FUNCTION_BLOCK FB_System_RND_HVAC
VAR_IN_OUT
	// Hold a reference to MBMaster - may need to share this with other dosing machines if only 1 x RS485 card is used for both
	{attribute 'OPC.UA.DA' := '0'}
  	{attribute 'OPC.UA.DA.StructuredType' := '0'}
	fbModbusManager: 	FB_ModbusManager;    // We can read 32 registers using one query
END_VAR

VAR
	bFirstRun: BOOL := TRUE;
	bResetTimer: BOOL := TRUE;
	tgModReadAdaptorStatus: R_TRIG;
	
	
	nModbusID: INT := 1;
	nNumberHVACUnits: INT := 13;
	
	stModReadAdaptorStatus: 				ST_Modbus_ReadRequest;
	
	stModReadIndoorUnitConnStatus: 			ST_Modbus_ReadRequest;
	stModReadIndoorUnitCommsStatus: 		ST_Modbus_ReadRequest;
	stModReadIndoorUnitSetpoits: 			ARRAY[1..13] OF ST_Modbus_ReadRequest;
	stModReadIndoorUnitPower: 				ARRAY[1..13] OF ST_Modbus_ReadRequest;
	
	stModWriteaAdaptorStatus:				ST_Modbus_WriteRequest;
	stModWriteIndoorRoom:					ST_Modbus_WriteRequest;
	stModWriteIndoorSetpoint_R6:			ST_Modbus_WriteRequest;
	stModWriteIndoorSetpoint_R7:			ST_Modbus_WriteRequest;
	stModWriteIndoorSetpoint_R8:			ST_Modbus_WriteRequest;
	stModWriteIndoorSetpoint_R9:			ST_Modbus_WriteRequest;
	stModWriteIndoorControlPower:			ARRAY[1..13] OF ST_Modbus_WriteRequest;
	stModWriteIndoorControlSetpoint:		ARRAY[1..13] OF ST_Modbus_WriteRequest;
	
	bRoom7or9: BOOL := FALSE;
	nRoomNumber: UINT := 6;
	
	fbTON_DataRefresh: TON := (PT := T#1m, IN := FALSE);
	
	// delete this after commissioning (used for testing)
	modWrite: R_TRIG;
	stModWrite: ST_Modbus_WriteRequest;
	
		// delete this after commissioning (used for testing)
	modRead: 	R_TRIG;
	stModRead: 	ST_Modbus_ReadRequest;
END_VAR

VAR_OUTPUT
	{attribute 'OPC.UA.DA' := '1'}
  	{attribute 'OPC.UA.DA.StructuredType' := '1'}
	fbRND_HVAC: ARRAY[1..13] OF FB_HVAC_RND_Indoor_Unit;
	
	
	i: INT := 0;
	
END_VAR

IF bFirstRun THEN
	devices_init();
	bFirstRun := FALSE;
	initModRequests();
	
	fbModbusManager.addRequest_Write(WriteRequest := ADR(stModWriteaAdaptorStatus));
	fbModbusManager.addRequest_Write(WriteRequest := ADR(stModWriteIndoorRoom));
END_IF

IF bResetTimer THEN
	fbTON_DataRefresh(IN := TRUE);
	bResetTimer := FALSE;
END_IF

fbTON_DataRefresh();
scanInputs();

IF fbTON_DataRefresh.Q THEN
	//fbModbusManager.addRequest_Read(ReadRequest := ADR(stModReadAdaptorStatus));
	//fbModbusManager.addRequest_Read(ReadRequest := ADR(stModReadIndoorUnitConnStatus));
	//fbModbusManager.addRequest_Read(ReadRequest := ADR(stModReadIndoorUnitCommsStatus));
	CASE nRoomNumber OF
		6:
			stModWriteIndoorSetpoint_R6.WriteRegVals[1] := INT_TO_WORD(REAL_TO_INT(Inputs.HVAC_RND[6].Setpoint * 10));
			fbModbusManager.addRequest_Write(WriteRequest := ADR(stModWriteIndoorSetpoint_R6));		
			nRoomNumber := 7;
	
		7:
			stModWriteIndoorSetpoint_R7.WriteRegVals[1] := INT_TO_WORD(REAL_TO_INT(Inputs.HVAC_RND[7].Setpoint * 10));
			fbModbusManager.addRequest_Write(WriteRequest := ADR(stModWriteIndoorSetpoint_R7));
			nRoomNumber := 8;
			
		8:
			stModWriteIndoorSetpoint_R8.WriteRegVals[1] := INT_TO_WORD(REAL_TO_INT(Inputs.HVAC_RND[8].Setpoint * 10));
			fbModbusManager.addRequest_Write(WriteRequest := ADR(stModWriteIndoorSetpoint_R8));
			nRoomNumber := 9;	
		
		9:
			stModWriteIndoorSetpoint_R9.WriteRegVals[1] := INT_TO_WORD(REAL_TO_INT(Inputs.HVAC_RND[9].Setpoint * 10));
			fbModbusManager.addRequest_Write(WriteRequest := ADR(stModWriteIndoorSetpoint_R9));
			nRoomNumber := 6;		
			
	END_CASE
	
	(*
	IF bRoom7or9 THEN
			stModWriteIndoorSetpoint_R7.WriteRegVals[1] := INT_TO_WORD(REAL_TO_INT(Inputs.HVAC_RND[7].Setpoint * 10));
			fbModbusManager.addRequest_Write(WriteRequest := ADR(stModWriteIndoorSetpoint_R7));
			bRoom7or9 := FALSE;
	ELSE
			stModWriteIndoorSetpoint_R9.WriteRegVals[1] := INT_TO_WORD(REAL_TO_INT(Inputs.HVAC_RND[9].Setpoint * 10));
			fbModbusManager.addRequest_Write(WriteRequest := ADR(stModWriteIndoorSetpoint_R9));
			bRoom7or9 := TRUE;
	END_IF
	*)

	

	
	//FOR i := 1 TO 13 DO
		//fbModbusManager.addRequest_Read(ReadRequest := ADR(stModReadIndoorUnitSetpoits[i]));
		//fbModbusManager.addRequest_Read(ReadRequest := ADR(stModReadIndoorUnitPower[i]));
		//fbModbusManager.addRequest_Write(WriteRequest := ADR(stModWriteIndoorControlPower));
		//fbModbusManager.addRequest_Write(WriteRequest := ADR(stModWriteIndoorControlSetpoint));
	//END_FOR
	
	fbTON_DataRefresh(IN := FALSE);
	bResetTimer := TRUE;
END_IF


modRead();
IF modRead.Q THEN
	fbModbusManager.addRequest_Read_Priority(ReadRequest := ADR(stModRead));
END_IF


modWrite();
IF modWrite.Q THEN
	fbModbusManager.addRequest_Write(WriteRequest := ADR(stModWrite));
END_IF

devices_update();

METHOD devices_init : BOOL
VAR_INPUT
END_VAR
(*
aHVAC_IndoorUnits[1] := ADR(fbRND1_HVAC);
aHVAC_IndoorUnits[2] := ADR(fbRND2_HVAC);
aHVAC_IndoorUnits[3] := ADR(fbRND3_HVAC);
aHVAC_IndoorUnits[4] := ADR(fbRND4_HVAC);
aHVAC_IndoorUnits[5] := ADR(fbRND5_HVAC);
aHVAC_IndoorUnits[6] := ADR(fbRND6_HVAC);
aHVAC_IndoorUnits[7] := ADR(fbRND7_HVAC);
aHVAC_IndoorUnits[8] := ADR(fbRND8_HVAC);
aHVAC_IndoorUnits[9] := ADR(fbRND9_HVAC);
aHVAC_IndoorUnits[10] := ADR(fbRND10_HVAC);
aHVAC_IndoorUnits[11] := ADR(fbRND11_HVAC);
aHVAC_IndoorUnits[12] := ADR(fbRND12_HVAC);

*)
END_METHOD

METHOD devices_update : BOOL
VAR_INPUT
END_VAR
(*
FOR i := 1 TO 13 DO
	fbRND_HVAC[i].bOnOff_1_0 := 	stModReadIndoorUnitPower[i].ReadRegsVals[1].0;
	fbRND_HVAC[1].nSetpoint_RO := 	WORD_TO_REAL(stModReadIndoorUnitSetpoits[i].ReadRegsVals[1])/10;
	
END_FOR

fbRND_HVAC[1].bConnectionStatus := stModReadIndoorUnitConnStatus.ReadRegsVals[1].0;
fbRND_HVAC[2].bConnectionStatus := stModReadIndoorUnitConnStatus.ReadRegsVals[1].1;
fbRND_HVAC[3].bConnectionStatus := stModReadIndoorUnitConnStatus.ReadRegsVals[1].2;
fbRND_HVAC[4].bConnectionStatus := stModReadIndoorUnitConnStatus.ReadRegsVals[1].3;
fbRND_HVAC[5].bConnectionStatus := stModReadIndoorUnitConnStatus.ReadRegsVals[1].4;
fbRND_HVAC[6].bConnectionStatus := stModReadIndoorUnitConnStatus.ReadRegsVals[1].5;
fbRND_HVAC[7].bConnectionStatus := stModReadIndoorUnitConnStatus.ReadRegsVals[1].6;
fbRND_HVAC[8].bConnectionStatus := stModReadIndoorUnitConnStatus.ReadRegsVals[1].7;
fbRND_HVAC[9].bConnectionStatus := stModReadIndoorUnitConnStatus.ReadRegsVals[1].8;
fbRND_HVAC[10].bConnectionStatus := stModReadIndoorUnitConnStatus.ReadRegsVals[1].9;
fbRND_HVAC[11].bConnectionStatus := stModReadIndoorUnitConnStatus.ReadRegsVals[1].10;
fbRND_HVAC[12].bConnectionStatus := stModReadIndoorUnitConnStatus.ReadRegsVals[1].11;
fbRND_HVAC[13].bConnectionStatus := stModReadIndoorUnitConnStatus.ReadRegsVals[1].12;

fbRND_HVAC[1].bCommsStatus := stModReadIndoorUnitCommsStatus.ReadRegsVals[1].0;
fbRND_HVAC[2].bCommsStatus := stModReadIndoorUnitCommsStatus.ReadRegsVals[1].1;
fbRND_HVAC[3].bCommsStatus := stModReadIndoorUnitCommsStatus.ReadRegsVals[1].2;
fbRND_HVAC[4].bCommsStatus := stModReadIndoorUnitCommsStatus.ReadRegsVals[1].3;
fbRND_HVAC[5].bCommsStatus := stModReadIndoorUnitCommsStatus.ReadRegsVals[1].4;
fbRND_HVAC[6].bCommsStatus := stModReadIndoorUnitCommsStatus.ReadRegsVals[1].5;
fbRND_HVAC[7].bCommsStatus := stModReadIndoorUnitCommsStatus.ReadRegsVals[1].6;
fbRND_HVAC[8].bCommsStatus := stModReadIndoorUnitCommsStatus.ReadRegsVals[1].7;
fbRND_HVAC[9].bCommsStatus := stModReadIndoorUnitCommsStatus.ReadRegsVals[1].8;
fbRND_HVAC[10].bCommsStatus := stModReadIndoorUnitCommsStatus.ReadRegsVals[1].9;
fbRND_HVAC[11].bCommsStatus := stModReadIndoorUnitCommsStatus.ReadRegsVals[1].10;
fbRND_HVAC[12].bCommsStatus := stModReadIndoorUnitCommsStatus.ReadRegsVals[1].11;
fbRND_HVAC[13].bCommsStatus := stModReadIndoorUnitCommsStatus.ReadRegsVals[1].12;
*)
END_METHOD

METHOD FB_init : BOOL
VAR_INPUT
	bInitRetains : BOOL; // if TRUE, the retain variables are initialized (warm start / cold start)
	bInCopyCode : BOOL;  // if TRUE, the instance afterwards gets moved into the copy code (online change)
	
	ModbusID: UINT;
END_VAR
nModbusID := ModbusID;
END_METHOD

METHOD initModRequests : BOOL
VAR_INPUT
END_VAR

stModReadAdaptorStatus.SlaveAddress := 1;
stModReadAdaptorStatus.AdrFirstSlaveRegisterRead := 0;
stModReadAdaptorStatus.QtyWordsToRead := 1;

stModReadIndoorUnitConnStatus.SlaveAddress := 1;
stModReadIndoorUnitConnStatus.AdrFirstSlaveRegisterRead := 1;
stModReadIndoorUnitConnStatus.QtyWordsToRead := 1;

stModReadIndoorUnitCommsStatus.SlaveAddress := 1;
stModReadIndoorUnitCommsStatus.AdrFirstSlaveRegisterRead := 5;
stModReadIndoorUnitCommsStatus.QtyWordsToRead := 1;

stModWriteaAdaptorStatus.SlaveAddress := 1;
stModWriteaAdaptorStatus.AdrFirstSlaveRegisterWrite := 1;
stModWriteaAdaptorStatus.QtyWordsToWrite := 1;
stModWriteaAdaptorStatus.WriteRegVals[1] := 32768; // turn modbus comms on

stModWriteIndoorRoom.SlaveAddress := 1;
stModWriteIndoorRoom.AdrFirstSlaveRegisterWrite := 2018;
stModWriteIndoorRoom.QtyWordsToWrite := 1;
stModWriteIndoorRoom.WriteRegVals[1] := 1889;

stModWriteIndoorSetpoint_R6.SlaveAddress := 1;
stModWriteIndoorSetpoint_R6.AdrFirstSlaveRegisterWrite := 2017;
stModWriteIndoorSetpoint_R6.QtyWordsToWrite := 1;

stModWriteIndoorSetpoint_R7.SlaveAddress := 1;
stModWriteIndoorSetpoint_R7.AdrFirstSlaveRegisterWrite := 2020;
stModWriteIndoorSetpoint_R7.QtyWordsToWrite := 1;

stModWriteIndoorSetpoint_R8.SlaveAddress := 1;
stModWriteIndoorSetpoint_R8.AdrFirstSlaveRegisterWrite := 2023;
stModWriteIndoorSetpoint_R8.QtyWordsToWrite := 1;

stModWriteIndoorSetpoint_R9.SlaveAddress := 1;
stModWriteIndoorSetpoint_R9.AdrFirstSlaveRegisterWrite := 2026;
stModWriteIndoorSetpoint_R9.QtyWordsToWrite := 1;


FOR i := 1 TO nNumberHVACUnits DO
	stModReadIndoorUnitSetpoits[i].SlaveAddress := 1;
	stModReadIndoorUnitSetpoits[i].AdrFirstSlaveRegisterRead := 2002 + ((i-1) * 6);
	stModReadIndoorUnitSetpoits[i].QtyWordsToRead := 1;
	
	stModReadIndoorUnitPower[i].SlaveAddress := 1;
	stModReadIndoorUnitPower[i].AdrFirstSlaveRegisterRead := 2000 + ((i-1) * 6);
	stModReadIndoorUnitPower[i].QtyWordsToRead := 1;
	
	stModWriteIndoorControlPower[i].SlaveAddress := 1;
	stModWriteIndoorControlPower[i].AdrFirstSlaveRegisterWrite := 2000 + ((i-1)*3);
	stModWriteIndoorControlPower[i].QtyWordsToWrite := 1;
	
	stModWriteIndoorControlSetpoint[i].SlaveAddress := 1;
	stModWriteIndoorControlSetpoint[i].AdrFirstSlaveRegisterWrite := 2002 + + ((i-1)*3);
	stModWriteIndoorControlSetpoint[i].QtyWordsToWrite := 1;
	
END_FOR
END_METHOD

METHOD scanInputs : BOOL
VAR_INPUT
END_VAR
FOR i := 1 TO nNumberHVACUnits DO
	IF Inputs.HVAC_RND[i].Power THEN
		stModWriteIndoorControlPower[i].WriteRegVals[1] := 1;
	ELSE
		stModWriteIndoorControlPower[i].WriteRegVals[1] := 0;
	END_IF
	//stModWriteIndoorControlPower[i].WriteRegVals[1] := BOOL_TO_WORD(Inputs.HVAC_RND[i].Power);
	stModWriteIndoorControlSetpoint[i].WriteRegVals[1] := (REAL_TO_INT(Inputs.HVAC_RND[i].Setpoint * 10.0));
	// stModWriteIndoorControlPower[i].WriteRegVals[i] := 2#0111001001100000 AND stModWriteIndoorControlPower[i].WriteRegVals[i]; // binary word includes mandatory fields (fan power / volume / control)
END_FOR
END_METHOD

END_FUNCTION_BLOCK

(* stored: Version 1.1.0.1, ProductVersion 3.1.4024.12
   POU FB_System_RND_HVAC: Id {e6b5ad06-e6be-4f9e-9253-204717a172fd}, SpecialFunc None
   Method devices_init: Id {914d674e-04ee-4858-a190-a7364df2abb6}
   Method devices_update: Id {fa73bb39-fd2c-4089-af24-99eb6cd5db8c}
   Method FB_init: Id {b333f4fd-8476-47a1-919d-1ed81e3b95ef}
   Method initModRequests: Id {7ac3b5a0-789d-420f-9fa8-08313aae926a}
   Method scanInputs: Id {361b0b9c-c3b5-4e26-9f66-6510310a3e15} *)
